// TIA Portal V20 export
VAR_GLOBAL   // PLC tag table "Fixture"
END_VAR
VAR_GLOBAL CONSTANT   // user constants
   X : USInt := 1;
   Y : USInt := 2;
   Z : USInt := 3;
   G : USInt := 4;
END_VAR
